# EPICS autosave request: dexelaApp/Db/Dexela_settings.req
$(P)$(R)DEXBinningMode
$(P)$(R)DEXCorrectionsDir
$(P)$(R)DEXNumOffsetFrames
$(P)$(R)DEXUseOffset
$(P)$(R)DEXOffsetFile
$(P)$(R)DEXOffsetConstant
$(P)$(R)DEXNumGainFrames
$(P)$(R)DEXUseGain
$(P)$(R)DEXGainFile
$(P)$(R)DEXUseDefectMap
$(P)$(R)DEXDefectMapFile
